RoboDK station: painting.rdk

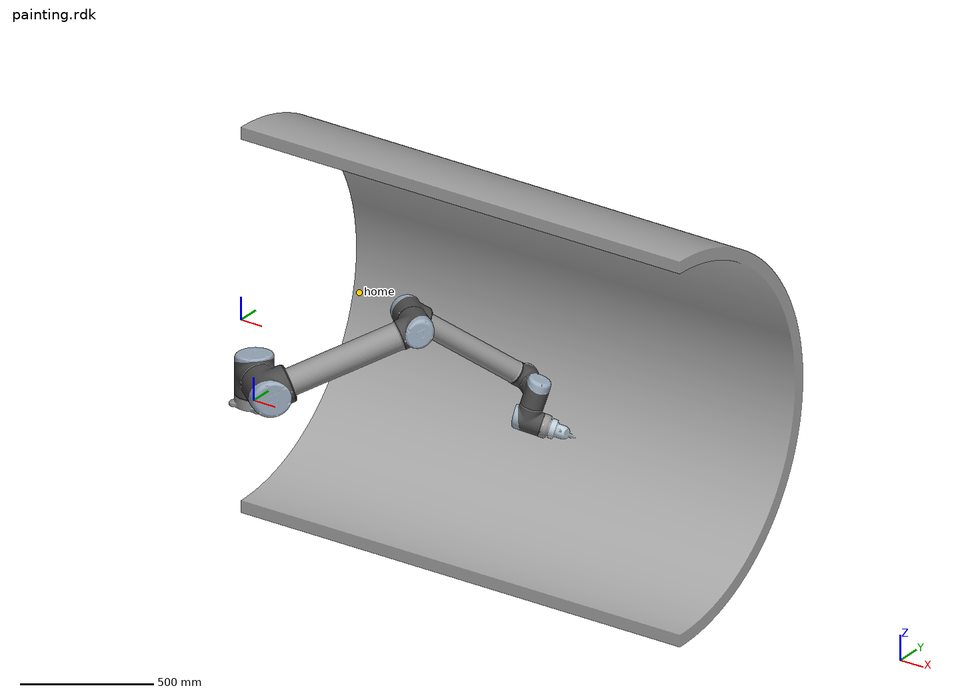
[picture v0: the station drawn from its stored meshes, robots at their saved joint values, targets as dots, program paths as lines]
Station painting. Poses are relative to the parent item; angles as X-Y-Z fixed-axis rotations.
  - frame UR10 Base at (0, 0, 0) mm
    - robot UR10: 6 axes, payload 10 kg, reach 1300 mm, repeatability 0.1 mm, weight 28.9 kg
        modified DH rows (alpha deg, a mm, theta deg, d mm): 0, 0, 0, 118; 90, 0, 180, 0; 0, 612.7, 0, 0; 0, 571.6, 0, 163.9; -90, 0, 0, 115.7; 90, 0, 180, 92.2
        joint limits [-360, -360, -360, -360, -360, -360] to [360, 360, 360, 360, 360, 360]; home [0, -90, 90, 0, 90, 0]; saved at [-309.799, 198.283, 306.209, 197.373, -66.274, 66.517]
      - tool Pencil, TCP at (1.16, -82.2, 101.78) mm, rotated rx 0 ry -60 rz 90 deg, size 74.9 x 125 x 107.3 mm
  - frame paintframe at (-200, 200, 200) mm
    - target home (Cartesian target) at (400, 200, 143.37) mm; joints [-256.628, 252.981, 228.847, 170.003, 32.59, 244.571] of UR10
    - object cylindar at (0, 0, 0) mm, size 2000 x 800 x 1600 mm, geometry from cylindar.stl
  - Python program main (listed below)

--- Python program main ---
# Type help("robolink") or help("robodk") for more information
# Press F5 to run the script
# Note: you do not need to keep a copy of this file, your python script is saved with the station
from robolink import *    # API to communicate with RoboDK
from robodk import *      # basic matrix operations
RL = Robolink()

# Notify user:
print('A Matlab version of this API is available in C:/RoboDK/Matlab/\n')
print('The API is also available in C#\n')
print('To edit this program:\nright click on the Python program, then, select "Edit Python script"\n')


import math

import numpy as np

def vectors2matrix(A,B):
   #A starting vector
   #B ending vector
   #returns: 3x3 matrix to rotate A to B

   rcos = np.dot(A, B)
   C = np.cross(A, B)
   rsin = np.linalg.norm(C)
   C = C/rsin

   u=C[0]
   v=C[1]
   w=C[2]
   R=np.array([[rcos + u*u*(1-rcos),  -w * rsin + u*v*(1-rcos), v * rsin + u*w*(1-rcos)],
                      [ w * rsin + v*u*(1-rcos), rcos + v*v*(1-rcos), -u * rsin + v*w*(1-rcos)],
                      [-v * rsin + w*u*(1-rcos), u * rsin + w*v*(1-rcos), rcos + w*w*(1-rcos)]])

   return(R)

def point2matrix(point):
    matrix_opposite = np.array([[-1,  0,  0],
                     [ 0, -1,  0],
                     [ 0,  0, -1]])
    start_vector = np.array([0, 0, 1])
    direction = np.dot(np.array([point[3], point[4], point[5]]), matrix_opposite)
    rotation_matrix = vectors2matrix(start_vector, direction)
    four_by_four = np.zeros((4,4))
    four_by_four[:3, :3]=rotation_matrix

    four_by_four[0][3]=point[0]
    four_by_four[1][3]=point[1]
    four_by_four[2][3]=point[2]
    four_by_four[3][3]=1
    return four_by_four


def matrix2pose(matrix):
    pose = Mat(4,4)
    for j in range(4):
        for i in range(4):
            pose[i,j] = matrix[i][j]
    return pose

def point2pose(point, matrix_more_change=None):
    m = point2matrix(point)
#    print("m:")
#    print(m)
    if matrix_more_change is None:
        p = matrix2pose(m)
    else:
        new_m = np.dot(m, matrix_more_change)
        p = matrix2pose(new_m)
#    print("p:")
#    print(p)
    return p

import numpy as np
points = np.genfromtxt ('C:\\Users\\Admin\\Documents\\VR_painting\\robotics\\test\\curves\\cylindar.csv', delimiter=",")

# Program example:
item = RL.Item('base')
if item.Valid():
    print('Item selected: ' + item.Name())
    print('Item posistion: ' + repr(item.Pose()))

#print('Items in the station:')
#itemlist = RL.ItemList()
#print(itemlist)

robot = RL.Item('UR10')
baseFrame = RL.Item('UR10 Base')
paintFrame = RL.Item('paintframe')

# get the home target and the welding targets:
robot.setFrame(paintFrame)
home = RL.Item('home')
#poseref = home.Pose()

#print('Home posistion: ' + repr(home.Pose()))
robot.MoveJ(home)

offset = np.array([[1.0, 0.0, 0.0, 0.0], [0.0, 1.0, 0.0, 0.0],[0.0, 0.0, 1.0, -5], [0.0, 0.0, 0.0, 1.0]])
distance_start = np.array([[1.0, 0.0, 0.0, 0.0],[0.0, 1.0, 0.0, 0.0],[0.0, 0.0, 1.0, -5.0], [0.0, 0.0, 0.0, 1.0]])
distance_retreat = np.array([[1.0, 0.0, 0.0, 0.0], [0.0, 1.0, 0.0, 0.0], [0.0, 0.0, 1.0, -5.0], [0.0, 0.0, 0.0, 1.0]])
for i in range(np.size(points,0)-1):
    print("move to ready position")
    p0 = point2pose(points[i], distance_start)
    print(p0)
    robot.MoveJ(p0)

    print("move to first point edge")
    p1 = point2pose(points[i], offset)
    robot.MoveJ(p1)

    print("move to second point on edge")
    p2 = point2pose(points[i+1], offset)
    robot.MoveL(p2)

    p3 = point2pose(points[i+1], distance_retreat)
    print("move to retreat position")
    print(p3)
    robot.MoveJ(p3)

robot.MoveJ(home)

#raise Exception('Program not edited.')


#for i in range(7):
#    ang = i*2*pi/6 #angle: 0, 60, 120, ...
#    #posei = poseref*rotz(ang)*transl(200,0,0)*rotz(-ang)
#    posei = poseref*rotz(ang)*transl(100,0,0)*rotz(-ang)
#    print(posei.__str__)
#    robot.MoveL(posei)
